{attribute 'qualified_only'}
VAR_GLOBAL
	RunningStates : RunningStates :=RunningStates.Preparation;
	CheckPrint : BOOL := FALSE;
	Layer1Good : BOOL := FALSE;
	PrintingStates: PrintingStates:=PrintingStates.PrepareModel;
	EntryPrint:BOOL:=TRUE;
	
END_VAR

(* stored: Version 1.1.0.1, ProductVersion 3.1.4024.15
   GVL GVL: Id {f0f7fe03-104c-4ac5-8c8b-0428b6b36959} *)
